FUNCTION FC_DT_TO_ISO8610 : STRING(39)
VAR_INPUT
	I_DT					: REFERENCE TO DT;
END_VAR

FC_DT_TO_ISO8610 := SYSTEMTIME_TO_ISO8601(DT_TO_SYSTEMTIME(I_DT), 0, FALSE, 0);

END_FUNCTION

(* stored: Version 1.1.0.1, ProductVersion 3.1.4024.13
   POU FC_DT_TO_ISO8610: Id {060dd33e-0ba9-47f0-afda-12aac293f6a8}, SpecialFunc None *)
